{attribute 'pack_mode' := '1'} 
TYPE ASCF_CC_OPCUACS_Reader_Temp_Real :
STRUCT
	stReadListReturnInfo	: ARRAY [1..2] OF ST_UAReadListReturnInfo;
	QC		: BYTE	:= 16#00;
	Value	: REAL	:= 0.0;
END_STRUCT
END_TYPE

(* stored: Version 1.1.0.1, ProductVersion 3.1.4026.4
   DUT ASCF_CC_OPCUACS_Reader_Temp_Real: Id {0fd99285-5ee9-4f6a-9d1b-80c54eceb9d6} *)
